Yaskawa INFORM job: SVETS2.JBI

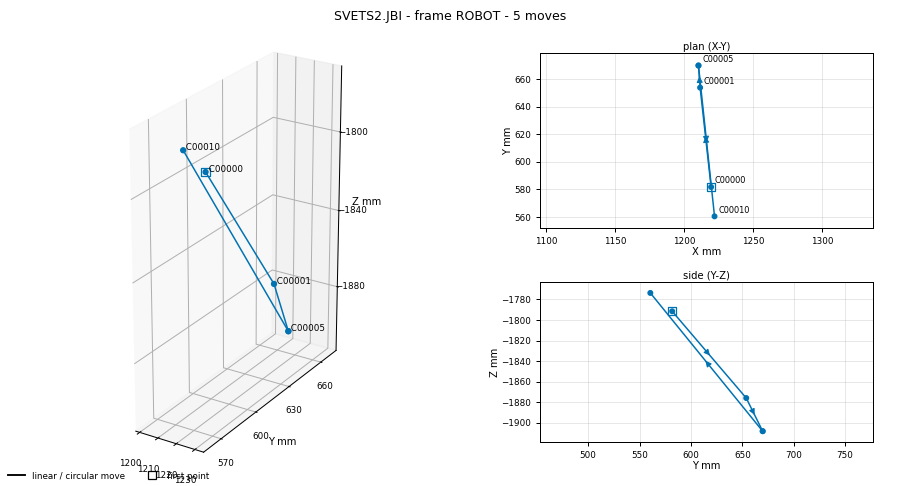
[picture p0: tool path of SVETS2.JBI in frame ROBOT, 5 of 5 moves have a stored position in this frame; points joined in program order, loops and branches not executed]
/JOB
//NAME SVETS2
///FOLDERNAME INNE
//POS
///NPOS 11,11,0,0,0,0
///TOOL 0
///POSTYPE ROBOT
///RECTAN
///RCONF 0,0,0,0,1,0,0,0,0,0,0,0,0,0,0,0,0,0,0,0,0,0,0,0
C00000=1219.583,581.792,-1791.458,40.6411,-1.1292,7.6176
C00001=1211.623,653.794,-1875.833,40.6405,-1.1296,7.6182
C00002=1211.623,653.794,-1875.833,40.6405,-1.1296,7.6182
C00003=1211.618,665.308,-1875.838,40.6404,-1.1289,7.6184
C00004=1211.607,653.793,-1888.348,40.6409,-1.1280,7.6177
C00005=1210.430,669.790,-1908.087,40.6410,-1.1296,7.6185
C00006=1210.406,664.661,-1844.435,40.6397,-1.1290,7.6184
C00007=1210.389,615.982,-1888.532,40.6537,-1.1257,7.6111
C00008=1210.742,663.101,-1893.795,40.6392,-1.1319,7.6205
C00009=1210.430,669.790,-1908.087,40.6410,-1.1296,7.6185
C00010=1222.064,560.522,-1773.626,40.6388,-1.1320,7.6208
///RCONF 0,0,0,0,0,0,0,0,0,0,0,0,0,0,0,0,0,0,0,0,0,0,0,0
BC00000=1.890,2751.820,818.150
BC00001=1.890,2751.820,818.150
BC00002=1.890,2751.820,818.150
BC00003=1.890,2751.820,818.150
BC00004=1.890,2751.820,818.150
BC00005=1.890,2751.820,818.150
BC00006=1.890,2751.820,818.150
BC00007=1.890,2751.820,818.148
BC00008=238.124,2751.820,818.150
BC00009=264.003,2759.033,818.898
BC00010=238.124,2751.820,818.150
//INST
///DATE 2023/10/04 15:16
///ATTR SC,RW,RJ
////FRAME ROBOT
///GROUP1 RB1,BS1
NOP
SFTOF
MOVL C00000 BC00000 V=150.0
MACRO1 MJ#(0) ARGF4
MOVL C00001 BC00001 V=75.0
REFP 4 C00002 BC00002
REFP 5 C00003 BC00003
REFP 6 C00004 BC00004
MOVL C00005 BC00005 V=75.0
REFP 1 C00006 BC00006
REFP 2 C00007 BC00007
REFP 3 C00008 BC00008
ARCON
WVON WEV#(1)
MOVL C00009 BC00009 V=7.5
WVOF
ARCOF
SFTOF
MOVL C00010 BC00010 V=150.0
END
